TYPE ST_JOB_STATE :
STRUCT
  State         : E_JOB_STATE;
END_STRUCT
END_TYPE

(* stored: Version 1.1.0.1
   DUT ST_JOB_STATE: Id {37274462-6f15-4434-9ce7-677e59bcf0fd} *)
